{attribute 'qualified_only'}
VAR_GLOBAL
	//metering signals
		MeteringSignals : feederMeteringStruct;
END_VAR

(* stored: Version 1.1.0.1, ProductVersion 3.1.4024.4
   GVL metering: Id {87ead626-b4bf-453b-8d89-b496fc9f482c} *)
